(* IEC 61131-3 sources: LabBench/POU/04_AlarmAndSafety/FB, 5 files *)

(* ---- FB_DiagnosticScenario.st ---- *)
(*==============================================================================
    Название:    FB_DiagnosticScenario
    Автор:
    Дата:        2025-04-30
    Версия:      1.0

    Описание:    Функциональный блок обработки сценариев диагностики
                 Анализирует состояние системы на предмет обнаружения сценариев
                 неисправностей, таких как "насос работает, но нет расхода" и т.п.
==============================================================================*)
FUNCTION_BLOCK FB_DiagnosticScenario
VAR_INPUT
    (* Входные сигналы состояния системы *)

    (* Состояние насосов *)
    bPump1Running: BOOL;           (* Насос 1 работает *)
    bPump2Running: BOOL;           (* Насос 2 работает *)
    rPump1Speed: REAL;             (* Скорость насоса 1 (%) *)
    rPump2Speed: REAL;             (* Скорость насоса 2 (%) *)

    (* Состояние клапанов *)
    rPropValvePosition: REAL;      (* Положение пропорционального клапана (%) *)
    bEMValveOpen: BOOL;            (* Состояние электромагнитного клапана *)

    (* Состояние нагревателя *)
    bHeaterOn: BOOL;               (* Нагреватель включен *)
    rHeaterPower: REAL;            (* Мощность нагревателя (%) *)

    (* Сигналы с датчиков *)

    (* Давление *)
    rPressureKIE2: REAL;           (* Давление в емкости КИЕ2 (кПа) *)
    bPressureKIE2Valid: BOOL;      (* Сигнал валиден *)

    rPressurePipe: REAL;           (* Давление в трубопроводе (кПа) *)
    bPressurePipeValid: BOOL;      (* Сигнал валиден *)

    rPressurePumpIn1: REAL;        (* Давление перед насосом 1 (кПа) *)
    bPressurePumpIn1Valid: BOOL;   (* Сигнал валиден *)

    rPressurePumpOut1: REAL;       (* Давление после насоса 1 (кПа) *)
    bPressurePumpOut1Valid: BOOL;  (* Сигнал валиден *)

    rPressurePumpIn2: REAL;        (* Давление перед насосом 2 (кПа) *)
    bPressurePumpIn2Valid: BOOL;   (* Сигнал валиден *)

    rPressurePumpOut2: REAL;       (* Давление после насоса 2 (кПа) *)
    bPressurePumpOut2Valid: BOOL;  (* Сигнал валиден *)

    (* Расход *)
    rFlowPumpOut1: REAL;           (* Расход после насоса 1 (л/мин) *)
    bFlowPumpOut1Valid: BOOL;      (* Сигнал валиден *)

    rFlowPumpOut2: REAL;           (* Расход после насоса 2 (л/мин) *)
    bFlowPumpOut2Valid: BOOL;      (* Сигнал валиден *)

    rFlowPipe: REAL;               (* Расход в трубопроводе (л/мин) *)
    bFlowPipeValid: BOOL;          (* Сигнал валиден *)

    (* Уровень *)
    rLevelKIE1: REAL;              (* Уровень в емкости КИЕ1 (мм) *)
    bLevelKIE1Valid: BOOL;         (* Сигнал валиден *)

    bLevelLow: BOOL;               (* Уровень низкий (поплавок) *)
    bLevelMid: BOOL;               (* Уровень средний (поплавок) *)
    bLevelHigh: BOOL;              (* Уровень высокий (поплавок) *)
    bLevelValid: BOOL;             (* Сигналы валидны *)

    (* Температура *)
    rTemperature: REAL;            (* Температура (°C) *)
    bTemperatureValid: BOOL;       (* Сигнал валиден *)

    (* Управление *)
    bReset: BOOL;                  (* Сброс сценариев *)
    bEnable: BOOL := TRUE;         (* Разрешение работы *)
END_VAR

VAR_OUTPUT
    bAnyScenarioActive: BOOL;      (* Флаг наличия активных сценариев *)
    bBlockingRequired: BOOL;       (* Требуется блокировка *)
    bShutdownRequired: BOOL;       (* Требуется останов *)
    uiActiveScenarioCount: UINT;   (* Количество активных сценариев *)
    uiLastActiveScenarioIndex: UINT; (* Индекс последнего активного сценария *)
    dwActiveScenariosMask: DWORD;  (* Битовая маска активных сценариев *)
END_VAR

VAR
    (* Триггеры для обнаружения изменений *)
    rtPump1Running: R_TRIG;        (* Насос 1 запустился *)
    rtPump2Running: R_TRIG;        (* Насос 2 запустился *)
    rtHeaterOn: R_TRIG;            (* Нагреватель включился *)

    ftPump1Running: F_TRIG;        (* Насос 1 остановился *)
    ftPump2Running: F_TRIG;        (* Насос 2 остановился *)
    ftHeaterOn: F_TRIG;            (* Нагреватель выключился *)

    (* Таймеры для задержек обнаружения *)
    tonScenario1: TON;             (* Таймер для сценария 1 *)
    tonScenario2: TON;             (* Таймер для сценария 2 *)
    tonScenario3: TON;             (* Таймер для сценария 3 *)

    (* Локальные переменные *)
    uiCounter: UINT;               (* Счетчик для циклов *)

    (* Параметры сценариев *)
    rPump1DeltaP: REAL;            (* Перепад давления на насосе 1 *)
    rPump2DeltaP: REAL;            (* Перепад давления на насосе 2 *)

    (* Флаги обнаружения условий сценариев *)
    bPump1NoFlow: BOOL;            (* Условие "Насос 1 работает, но нет расхода" *)
    bPump2NoFlow: BOOL;            (* Условие "Насос 2 работает, но нет расхода" *)
    bPump1NoPressure: BOOL;        (* Условие "Насос 1 работает, но нет давления" *)
    bPump2NoPressure: BOOL;        (* Условие "Насос 2 работает, но нет давления" *)
    bPipeBlock: BOOL;              (* Условие "Блокировка в трубопроводе" *)
    bHeaterNoTempRise: BOOL;       (* Условие "Нагреватель включен, но температура не растет" *)
END_VAR

VAR CONSTANT
    (* Пороговые значения для обнаружения сценариев *)
    PUMP_MIN_SPEED: REAL := 10.0;          (* Минимальная скорость насоса (%) *)
    FLOW_THRESHOLD_LOW: REAL := 0.5;       (* Пороговое значение расхода (л/мин) *)
    PRESSURE_DELTA_MIN: REAL := 10.0;      (* Минимальный перепад давления (кПа) *)
    TEMPERATURE_RISE_MIN: REAL := 0.1;     (* Минимальный рост температуры (°C/мин) *)

    (* Времена задержек для обнаружения сценариев *)
    T_PUMP_NO_FLOW: TIME := T#5S;          (* Задержка для сценария "нет расхода" *)
    T_PUMP_NO_PRESSURE: TIME := T#3S;      (* Задержка для сценария "нет давления" *)
    T_HEATER_NO_TEMP: TIME := T#60S;       (* Задержка для сценария "нет роста температуры" *)
END_VAR

(* ======================================================================== *)
(* Основная логика функционального блока                                    *)
(* ======================================================================== *)

(* Обнаружение изменений состояния оборудования *)
rtPump1Running(CLK := bPump1Running);
rtPump2Running(CLK := bPump2Running);
rtHeaterOn(CLK := bHeaterOn);

ftPump1Running(CLK := bPump1Running);
ftPump2Running(CLK := bPump2Running);
ftHeaterOn(CLK := bHeaterOn);

(* Обработка команды сброса *)
IF bReset THEN
    (* Сброс всех сценариев *)
    FOR uiCounter := 1 TO MAX_SCENARIOS DO
        gaDiagScenarios[uiCounter].bActive := FALSE;
    END_FOR;

    (* Сброс таймеров *)
    tonScenario1(IN := FALSE);
    tonScenario2(IN := FALSE);
    tonScenario3(IN := FALSE);
END_IF;

(* Инициализация выходных переменных *)
bAnyScenarioActive := FALSE;
bBlockingRequired := FALSE;
bShutdownRequired := FALSE;
uiActiveScenarioCount := 0;
uiLastActiveScenarioIndex := 0;
dwActiveScenariosMask := 0;

(* ======================================================================== *)
(* Обнаружение условий для сценариев                                        *)
(* ======================================================================== *)

IF bEnable THEN

    (* Расчет параметров системы *)
    IF bPressurePumpIn1Valid AND bPressurePumpOut1Valid THEN
        rPump1DeltaP := rPressurePumpOut1 - rPressurePumpIn1;
    ELSE
        rPump1DeltaP := 0.0;
    END_IF;

    IF bPressurePumpIn2Valid AND bPressurePumpOut2Valid THEN
        rPump2DeltaP := rPressurePumpOut2 - rPressurePumpIn2;
    ELSE
        rPump2DeltaP := 0.0;
    END_IF;

    (* Условие "Насос 1 работает, но нет расхода" *)
    bPump1NoFlow := bPump1Running AND rPump1Speed > PUMP_MIN_SPEED AND
                    bFlowPumpOut1Valid AND rFlowPumpOut1 < FLOW_THRESHOLD_LOW;

    (* Условие "Насос 2 работает, но нет расхода" *)
    bPump2NoFlow := bPump2Running AND rPump2Speed > PUMP_MIN_SPEED AND
                    bFlowPumpOut2Valid AND rFlowPumpOut2 < FLOW_THRESHOLD_LOW;

    (* Условие "Насос 1 работает, но нет давления" *)
    bPump1NoPressure := bPump1Running AND rPump1Speed > PUMP_MIN_SPEED AND
                        bPressurePumpIn1Valid AND bPressurePumpOut1Valid AND
                        rPump1DeltaP < PRESSURE_DELTA_MIN;

    (* Условие "Насос 2 работает, но нет давления" *)
    bPump2NoPressure := bPump2Running AND rPump2Speed > PUMP_MIN_SPEED AND
                        bPressurePumpIn2Valid AND bPressurePumpOut2Valid AND
                        rPump2DeltaP < PRESSURE_DELTA_MIN;

    (* Условие "Блокировка в трубопроводе" *)
    bPipeBlock := bFlowPipeValid AND rFlowPipe < FLOW_THRESHOLD_LOW AND
                  bPressurePipeValid AND rPressurePipe > (rPressureKIE2 * 1.5);

    (* Условие "Нагреватель включен, но температура не растет" *)
    (* Требует дополнительной логики с отслеживанием изменения температуры во времени *)
    bHeaterNoTempRise := FALSE; (* Пока не реализовано *)

    (* ======================================================================== *)
    (* Обработка таймеров задержки обнаружения сценариев                       *)
    (* ======================================================================== *)

    (* Таймер для сценария "Насос 1 работает, но нет расхода" *)
    tonScenario1(IN := bPump1NoFlow, PT := T_PUMP_NO_FLOW);

    (* Таймер для сценария "Насос 2 работает, но нет расхода" *)
    tonScenario2(IN := bPump2NoFlow, PT := T_PUMP_NO_FLOW);

    (* Таймер для сценария "Нагреватель включен, но температура не растет" *)
    tonScenario3(IN := bHeaterNoTempRise, PT := T_HEATER_NO_TEMP);

    (* ======================================================================== *)
    (* Активация сценариев диагностики                                         *)
    (* ======================================================================== *)

    (* Сценарий 1: "Насос 1 работает, но нет расхода" *)
    IF tonScenario1.Q THEN
        gaDiagScenarios[1].bActive := TRUE;
        gaDiagScenarios[1].eType := DIAG_PUMP_NO_FLOW;
        gaDiagScenarios[1].wSourceID := PUMP1_ID;
        gaDiagScenarios[1].wDeviceID := PUMP1_ID;
        gaDiagScenarios[1].eBlockingLevel := DEVICE_BLOCKING;
        gaDiagScenarios[1].bRequireShutdown := FALSE;
        gaDiagScenarios[1].rValue1 := rPump1Speed;
        gaDiagScenarios[1].rValue2 := rFlowPumpOut1;
        gaDiagScenarios[1].wErrorCode := 16#0101;
        gaDiagScenarios[1].sMessage := 'Насос 1 работает, но нет расхода';
    END_IF;

    (* Сценарий 2: "Насос 2 работает, но нет расхода" *)
    IF tonScenario2.Q THEN
        gaDiagScenarios[2].bActive := TRUE;
        gaDiagScenarios[2].eType := DIAG_PUMP_NO_FLOW;
        gaDiagScenarios[2].wSourceID := PUMP2_ID;
        gaDiagScenarios[2].wDeviceID := PUMP2_ID;
        gaDiagScenarios[2].eBlockingLevel := DEVICE_BLOCKING;
        gaDiagScenarios[2].bRequireShutdown := FALSE;
        gaDiagScenarios[2].rValue1 := rPump2Speed;
        gaDiagScenarios[2].rValue2 := rFlowPumpOut2;
        gaDiagScenarios[2].wErrorCode := 16#0102;
        gaDiagScenarios[2].sMessage := 'Насос 2 работает, но нет расхода';
    END_IF;

    (* Сценарий 3: "Насос 1 работает, но нет давления" *)
    IF bPump1NoPressure THEN
        gaDiagScenarios[3].bActive := TRUE;
        gaDiagScenarios[3].eType := DIAG_PUMP_NO_PRESSURE;
        gaDiagScenarios[3].wSourceID := PUMP1_ID;
        gaDiagScenarios[3].wDeviceID := PUMP1_ID;
        gaDiagScenarios[3].eBlockingLevel := DEVICE_BLOCKING;
        gaDiagScenarios[3].bRequireShutdown := FALSE;
        gaDiagScenarios[3].rValue1 := rPump1Speed;
        gaDiagScenarios[3].rValue2 := rPump1DeltaP;
        gaDiagScenarios[3].wErrorCode := 16#0103;
        gaDiagScenarios[3].sMessage := 'Насос 1 работает, но нет давления';
    END_IF;

    (* Сценарий 4: "Насос 2 работает, но нет давления" *)
    IF bPump2NoPressure THEN
        gaDiagScenarios[4].bActive := TRUE;
        gaDiagScenarios[4].eType := DIAG_PUMP_NO_PRESSURE;
        gaDiagScenarios[4].wSourceID := PUMP2_ID;
        gaDiagScenarios[4].wDeviceID := PUMP2_ID;
        gaDiagScenarios[4].eBlockingLevel := DEVICE_BLOCKING;
        gaDiagScenarios[4].bRequireShutdown := FALSE;
        gaDiagScenarios[4].rValue1 := rPump2Speed;
        gaDiagScenarios[4].rValue2 := rPump2DeltaP;
        gaDiagScenarios[4].wErrorCode := 16#0104;
        gaDiagScenarios[4].sMessage := 'Насос 2 работает, но нет давления';
    END_IF;

    (* Сценарий 5: "Блокировка в трубопроводе" *)
    IF bPipeBlock THEN
        gaDiagScenarios[5].bActive := TRUE;
        gaDiagScenarios[5].eType := DIAG_PIPE_BLOCK;
        gaDiagScenarios[5].wSourceID := SYSTEM_ID;
        gaDiagScenarios[5].wDeviceID := 0;
        gaDiagScenarios[5].eBlockingLevel := SYSTEM_BLOCKING;
        gaDiagScenarios[5].bRequireShutdown := TRUE;
        gaDiagScenarios[5].rValue1 := rFlowPipe;
        gaDiagScenarios[5].rValue2 := rPressurePipe;
        gaDiagScenarios[5].wErrorCode := 16#0105;
        gaDiagScenarios[5].sMessage := 'Блокировка в трубопроводе';
    END_IF;

    (* Сценарий 6: "Нагреватель включен, но температура не растет" *)
    IF tonScenario3.Q THEN
        gaDiagScenarios[6].bActive := TRUE;
        gaDiagScenarios[6].eType := DIAG_HEATER_NO_TEMP_RISE;
        gaDiagScenarios[6].wSourceID := HEATER_ID;
        gaDiagScenarios[6].wDeviceID := HEATER_ID;
        gaDiagScenarios[6].eBlockingLevel := DEVICE_BLOCKING;
        gaDiagScenarios[6].bRequireShutdown := FALSE;
        gaDiagScenarios[6].rValue1 := rHeaterPower;
        gaDiagScenarios[6].rValue2 := rTemperature;
        gaDiagScenarios[6].wErrorCode := 16#0106;
        gaDiagScenarios[6].sMessage := 'Нагреватель включен, но температура не растет';
    END_IF;

    (* ======================================================================== *)
    (* Обработка результатов анализа сценариев                                 *)
    (* ======================================================================== *)

    (* Обработка всех сценариев *)
    FOR uiCounter := 1 TO MAX_SCENARIOS DO
        IF gaDiagScenarios[uiCounter].bActive THEN
            (* Сценарий активен *)
            bAnyScenarioActive := TRUE;
            uiActiveScenarioCount := uiActiveScenarioCount + 1;
            uiLastActiveScenarioIndex := uiCounter;

            (* Установка бита в маске активных сценариев (только для первых 32 сценариев) *)
            IF uiCounter <= 32 THEN
                dwActiveScenariosMask := dwActiveScenariosMask OR SHL(DWORD#1, uiCounter-1);
            END_IF;

            (* Проверка требований блокировки и останова *)
            IF gaDiagScenarios[uiCounter].eBlockingLevel <> NO_BLOCKING THEN
                bBlockingRequired := TRUE;
            END_IF;

            IF gaDiagScenarios[uiCounter].bRequireShutdown THEN
                bShutdownRequired := TRUE;
            END_IF;
        END_IF;
    END_FOR;
END_IF;

(* ---- FB_ErrorManager.st ---- *)
(*==============================================================================
    Название:    FB_ErrorManager
    Автор:
    Дата:        2025-04-28
    Версия:      1.0

    Описание:    Функциональный блок управления ошибками и блокировками
                 Обрабатывает ошибки различных категорий, управляет блокировками
                 оборудования и формирует сигналы для сигнальной лампы
==============================================================================*)
FUNCTION_BLOCK FB_ErrorManager
VAR_INPUT
    bResetAll: BOOL;                      (* Общий сброс всех ошибок *)
    bResetMeasurement: BOOL;              (* Сброс ошибок измерительной системы *)
    bResetPropValve: BOOL;                (* Сброс ошибок пропорционального клапана *)
    bResetEMValve: BOOL;                  (* Сброс ошибок электромагнитного клапана *)
    bResetPump1: BOOL;                    (* Сброс ошибок насоса 1 *)
    bResetPump2: BOOL;                    (* Сброс ошибок насоса 2 *)
END_VAR

VAR_OUTPUT
    bAnyError: BOOL;                      (* Флаг наличия любых ошибок *)
    bSystemBlocking: BOOL;                (* Флаг полной блокировки системы *)
    eLampMode: E_LampBlinkMode;           (* Режим работы сигнальной лампы *)
    dwActiveErrorMask: DWORD;             (* Битовая маска активных ошибок *)

    (* Блокировки устройств *)
    bPropValveBlocking: BOOL;             (* Блокировка пропорционального клапана *)
    bEMValveBlocking: BOOL;               (* Блокировка электромагнитного клапана *)
    bPump1Blocking: BOOL;                 (* Блокировка насоса 1 *)
    bPump2Blocking: BOOL;                 (* Блокировка насоса 2 *)
END_VAR

VAR
    (* Локальные переменные *)
    uiCounter: UINT;                      (* Счетчик для циклов *)
    bHasErrorCategory: ARRAY[0..4] OF BOOL; (* Флаги наличия ошибок по категориям *)
END_VAR

(* ======================================================================== *)
(* Основная логика функционального блока                                    *)
(* ======================================================================== *)

(* Обработка команд сброса ошибок *)
IF bResetAll THEN
    (* Сброс всех ошибок *)
    FOR uiCounter := 1 TO MAX_ERRORS DO
        gaBlockingErrors[uiCounter].bActive := FALSE;
    END_FOR;
ELSE
    (* Выборочный сброс ошибок *)
    IF bResetMeasurement THEN
        (* Сброс ошибок измерительной системы *)
        FOR uiCounter := 1 TO MAX_ERRORS DO
            IF gaBlockingErrors[uiCounter].eCategory = ERROR_MEASUREMENT THEN
                gaBlockingErrors[uiCounter].bActive := FALSE;
            END_IF;
        END_FOR;
    END_IF;

    IF bResetPropValve THEN
        (* Сброс ошибок пропорционального клапана *)
        FOR uiCounter := 1 TO MAX_ERRORS DO
            IF gaBlockingErrors[uiCounter].wDeviceID = PROP_VALVE_ID THEN
                gaBlockingErrors[uiCounter].bActive := FALSE;
            END_IF;
        END_FOR;
    END_IF;

    IF bResetEMValve THEN
        (* Сброс ошибок электромагнитного клапана *)
        FOR uiCounter := 1 TO MAX_ERRORS DO
            IF gaBlockingErrors[uiCounter].wDeviceID = EM_VALVE_ID THEN
                gaBlockingErrors[uiCounter].bActive := FALSE;
            END_IF;
        END_FOR;
    END_IF;

    IF bResetPump1 THEN
        (* Сброс ошибок насоса 1 *)
        FOR uiCounter := 1 TO MAX_ERRORS DO
            IF gaBlockingErrors[uiCounter].wDeviceID = PUMP1_ID THEN
                gaBlockingErrors[uiCounter].bActive := FALSE;
            END_IF;
        END_FOR;
    END_IF;

    IF bResetPump2 THEN
        (* Сброс ошибок насоса 2 *)
        FOR uiCounter := 1 TO MAX_ERRORS DO
            IF gaBlockingErrors[uiCounter].wDeviceID = PUMP2_ID THEN
                gaBlockingErrors[uiCounter].bActive := FALSE;
            END_IF;
        END_FOR;
    END_IF;
END_IF;

(* Сброс флагов *)
bAnyError := FALSE;
bSystemBlocking := FALSE;
dwActiveErrorMask := 0;
bPropValveBlocking := FALSE;
bEMValveBlocking := FALSE;
bPump1Blocking := FALSE;
bPump2Blocking := FALSE;

(* Сброс флагов категорий ошибок *)
FOR uiCounter := 0 TO 4 DO
    bHasErrorCategory[uiCounter] := FALSE;
END_FOR;

(* Обработка всех ошибок *)
FOR uiCounter := 1 TO MAX_ERRORS DO
    IF gaBlockingErrors[uiCounter].bActive THEN
        (* Ошибка активна *)
        bAnyError := TRUE;

        (* Установка бита в маске активных ошибок (только для первых 32 ошибок) *)
        IF uiCounter <= 32 THEN
            dwActiveErrorMask := dwActiveErrorMask OR SHL(DWORD#1, uiCounter-1);
        END_IF;

        (* Отметка категории ошибки *)
        bHasErrorCategory[ENUM_TO_DINT(gaBlockingErrors[uiCounter].eCategory)] := TRUE;

        (* Обработка блокировок *)
        CASE gaBlockingErrors[uiCounter].eBlockingLevel OF
            SYSTEM_BLOCKING:
                (* Полная блокировка системы *)
                bSystemBlocking := TRUE;

            DEVICE_BLOCKING:
                (* Блокировка конкретного устройства *)
                CASE gaBlockingErrors[uiCounter].wDeviceID OF
                    PROP_VALVE_ID:
                        bPropValveBlocking := TRUE;

                    EM_VALVE_ID:
                        bEMValveBlocking := TRUE;

                    PUMP1_ID:
                        bPump1Blocking := TRUE;

                    PUMP2_ID:
                        bPump2Blocking := TRUE;
                END_CASE;
        END_CASE;
    END_IF;
END_FOR;

(* Определение режима работы сигнальной лампы *)
IF bAnyError THEN
    IF bHasErrorCategory[ENUM_TO_DINT(ERROR_MEASUREMENT)] THEN
        (* Ошибка измерения - быстрое мигание *)
        eLampMode := LAMP_FAST;
    ELSIF bHasErrorCategory[ENUM_TO_DINT(ERROR_COMMUNICATION)] THEN
        (* Ошибка связи - медленное мигание *)
        eLampMode := LAMP_SLOW;
    ELSIF bHasErrorCategory[ENUM_TO_DINT(ERROR_EQUIPMENT)] THEN
        (* Ошибка оборудования - постоянно горит *)
        eLampMode := LAMP_ON;
    ELSIF bHasErrorCategory[ENUM_TO_DINT(ERROR_PROCESS)] THEN
        (* Ошибка процесса - быстрое мигание *)
        eLampMode := LAMP_FAST;
    ELSE
        (* Неизвестная ошибка - постоянно горит *)
        eLampMode := LAMP_ON;
    END_IF;
ELSE
    (* Нет ошибок - лампа выключена *)
    eLampMode := LAMP_OFF;
END_IF;

(* ---- FB_LampController.st ---- *)
(*==============================================================================
    Название:    FB_LampController
    Автор:
    Дата:        2025-04-28
    Версия:      1.1

    Описание:    Функциональный блок управления сигнальной лампой
                 Генерирует сигналы для различных режимов работы лампы

                 Реализован как level-controlled (LCon) блок
==============================================================================*)
FUNCTION_BLOCK FB_LampController (* LCon *)
VAR_INPUT
    eMode: E_LampBlinkMode;               (* Режим работы лампы *)
    bEnable: BOOL := TRUE;                (* Разрешение работы *)
END_VAR

VAR_OUTPUT
    bOutput: BOOL;                        (* Выходной сигнал *)
END_VAR

VAR
    (* Таймеры для различных режимов мигания *)
    tonSlow: TON;                         (* Таймер медленного мигания (1 Гц) *)
    tonFast: TON;                         (* Таймер быстрого мигания (4 Гц) *)

    (* Состояния для различных режимов *)
    bSlowState: BOOL;                     (* Состояние медленного мигания *)
    bFastState: BOOL;                     (* Состояние быстрого мигания *)
END_VAR

VAR CONSTANT
    (* Константы времени для различных режимов *)
    T_SLOW: TIME := T#500MS;              (* Период для медленного мигания - 1 Гц *)
    T_FAST: TIME := T#125MS;              (* Период для быстрого мигания - 4 Гц *)
END_VAR

(* ======================================================================== *)
(* Основная логика функционального блока                                    *)
(* ======================================================================== *)

(* Генерация сигналов для различных режимов мигания *)
(* Медленное мигание - 1 Гц *)
tonSlow(IN := NOT tonSlow.Q, PT := T_SLOW);
IF tonSlow.Q THEN
    bSlowState := NOT bSlowState;
END_IF;

(* Быстрое мигание - 4 Гц *)
tonFast(IN := NOT tonFast.Q, PT := T_FAST);
IF tonFast.Q THEN
    bFastState := NOT bFastState;
END_IF;

(* Выбор режима мигания *)
IF bEnable THEN
    CASE eMode OF
        LAMP_OFF:
            bOutput := FALSE;

        LAMP_ON:
            bOutput := TRUE;

        LAMP_SLOW:
            bOutput := bSlowState;

        LAMP_FAST:
            bOutput := bFastState;

        ELSE
            (* По умолчанию - выключено *)
            bOutput := FALSE;
    END_CASE;
ELSE
    (* При отключенном блоке - выходной сигнал выключен *)
    bOutput := FALSE;
END_IF;

(* ---- FB_ShutdownSequencer.st ---- *)
(*==============================================================================
    Название:    FB_ShutdownSequencer
    Автор:
    Дата:        2025-04-30
    Версия:      1.0

    Описание:    Функциональный блок для управления последовательностью останова
                 Обеспечивает правильный порядок выключения оборудования
                 в штатном и аварийном режимах
==============================================================================*)
FUNCTION_BLOCK FB_ShutdownSequencer
VAR_IN_OUT
    stSequence: ST_ShutdownSequence;   (* Структура данных последовательности останова *)
END_VAR

VAR_INPUT
    bStartNormal: BOOL;                (* Запуск нормального останова *)
    bStartEmergency: BOOL;             (* Запуск аварийного останова *)
    bReset: BOOL;                      (* Сброс последовательности *)

    (* Состояние оборудования *)
    bHeaterOn: BOOL;                   (* Нагреватель включен *)
    rPump1Speed: REAL;                 (* Скорость насоса 1 (%) *)
    rPump2Speed: REAL;                 (* Скорость насоса 2 (%) *)
    rPropValvePosition: REAL;          (* Положение пропорционального клапана (%) *)
    bEMValveOpen: BOOL;                (* Состояние электромагнитного клапана *)
END_VAR

VAR_OUTPUT
    (* Команды управления оборудованием *)
    bHeaterOff: BOOL;                  (* Команда выключения нагревателя *)
    rPump1SpeedSetpoint: REAL;         (* Задание скорости насоса 1 (%) *)
    rPump2SpeedSetpoint: REAL;         (* Задание скорости насоса 2 (%) *)
    bPump1Stop: BOOL;                  (* Команда остановки насоса 1 *)
    bPump2Stop: BOOL;                  (* Команда остановки насоса 2 *)
    rPropValveSetpoint: REAL;          (* Задание положения пропорционального клапана (%) *)
    bEMValveClose: BOOL;               (* Команда закрытия электромагнитного клапана *)
END_VAR

VAR
    (* Триггеры *)
    rtStartNormal: R_TRIG;             (* Триггер запуска нормального останова *)
    rtStartEmergency: R_TRIG;          (* Триггер запуска аварийного останова *)
    rtReset: R_TRIG;                   (* Триггер сброса *)

    (* Таймеры *)
    tonStep: TON;                      (* Таймер текущего шага *)
    tonTimeout: TON;                   (* Таймер таймаута *)

    (* Локальные переменные *)
    tCurrentTime: TIME;                (* Текущее время *)
    tElapsedTime: TIME;                (* Прошедшее время *)
    rRateCalc: REAL;                   (* Расчетная скорость изменения *)
END_VAR

(* ======================================================================== *)
(* Основная логика функционального блока                                    *)
(* ======================================================================== *)

(* Обработка триггеров *)
rtStartNormal(CLK := bStartNormal);
rtStartEmergency(CLK := bStartEmergency);
rtReset(CLK := bReset);

(* Запуск последовательности останова *)
IF rtStartNormal.Q OR rtStartEmergency.Q THEN
    (* Инициализация последовательности *)
    stSequence.eCurrentStep := SHUTDOWN_INIT;
    stSequence.bInProgress := TRUE;
    stSequence.bEmergency := rtStartEmergency.Q;
    stSequence.bCompleted := FALSE;
    stSequence.bError := FALSE;
    stSequence.tStepStartTime := T#0S;

    (* Сброс таймеров *)
    tonStep(IN := FALSE);
    tonTimeout(IN := FALSE);
END_IF;

(* Сброс последовательности *)
IF rtReset.Q THEN
    (* Сброс всех параметров *)
    stSequence.eCurrentStep := SHUTDOWN_INIT;
    stSequence.bInProgress := FALSE;
    stSequence.bEmergency := FALSE;
    stSequence.bCompleted := FALSE;
    stSequence.bError := FALSE;
    stSequence.tStepStartTime := T#0S;

    (* Сброс таймеров *)
    tonStep(IN := FALSE);
    tonTimeout(IN := FALSE);

    (* Сброс выходов *)
    bHeaterOff := FALSE;
    rPump1SpeedSetpoint := 100.0;
    rPump2SpeedSetpoint := 100.0;
    bPump1Stop := FALSE;
    bPump2Stop := FALSE;
    rPropValveSetpoint := 100.0;
    bEMValveClose := FALSE;

    RETURN;
END_IF;

(* Обработка последовательности останова *)
IF stSequence.bInProgress THEN
    (* Отработка шагов последовательности *)
    CASE stSequence.eCurrentStep OF
        SHUTDOWN_INIT:
            (* Инициализация последовательности *)
            stSequence.tStepStartTime := T#0S;
            bHeaterOff := FALSE;
            bPump1Stop := FALSE;
            bPump2Stop := FALSE;
            bEMValveClose := FALSE;

            (* Переход к следующему шагу *)
            stSequence.eCurrentStep := SHUTDOWN_HEATER_OFF;

        SHUTDOWN_HEATER_OFF:
            (* Выключение нагревателя *)
            bHeaterOff := TRUE;

            (* Проверка выполнения шага *)
            IF NOT bHeaterOn THEN
                (* Нагреватель выключен - переход к следующему шагу *)
                stSequence.eCurrentStep := SHUTDOWN_PUMP_SLOWDOWN;
                tonStep(IN := FALSE);
            ELSE
                (* Ожидание выключения с таймаутом *)
                tonStep(IN := TRUE, PT := stSequence.tHeaterOffTimeout);
                IF tonStep.Q THEN
                    (* Таймаут - переход к следующему шагу с ошибкой *)
                    stSequence.eCurrentStep := SHUTDOWN_PUMP_SLOWDOWN;
                    stSequence.bError := TRUE;
                    tonStep(IN := FALSE);
                END_IF;
            END_IF;

        SHUTDOWN_PUMP_SLOWDOWN:
            (* Снижение скорости насосов *)
            IF stSequence.bEmergency THEN
                (* Аварийный останов - сразу к остановке насосов *)
                stSequence.eCurrentStep := SHUTDOWN_PUMP_STOP;
            ELSE
                (* Плавное снижение скорости насосов *)
                tonStep(IN := TRUE, PT := stSequence.tPumpSlowdownTime);

                (* Расчет скорости с учетом прошедшего времени *)
                rRateCalc := 100.0 - (TIME_TO_REAL(tonStep.ET) / TIME_TO_REAL(stSequence.tPumpSlowdownTime)) * 100.0;

                (* Установка скорости насосов *)
                rPump1SpeedSetpoint := MAX(0.0, rRateCalc);
                rPump2SpeedSetpoint := MAX(0.0, rRateCalc);

                (* Проверка завершения шага *)
                IF tonStep.Q THEN
                    (* Снижение скорости завершено - переход к остановке насосов *)
                    stSequence.eCurrentStep := SHUTDOWN_PUMP_STOP;
                    tonStep(IN := FALSE);
                END_IF;
            END_IF;

        SHUTDOWN_PUMP_STOP:
            (* Полная остановка насосов *)
            bPump1Stop := TRUE;
            bPump2Stop := TRUE;
            rPump1SpeedSetpoint := 0.0;
            rPump2SpeedSetpoint := 0.0;

            (* Проверка выполнения шага *)
            IF rPump1Speed <= 0.1 AND rPump2Speed <= 0.1 THEN
                (* Насосы остановлены - переход к следующему шагу *)
                stSequence.eCurrentStep := SHUTDOWN_VALVE_CLOSE;
                tonStep(IN := FALSE);
            ELSE
                (* Ожидание остановки с таймаутом *)
                tonStep(IN := TRUE, PT := stSequence.tPumpStopTimeout);
                IF tonStep.Q THEN
                    (* Таймаут - переход к следующему шагу с ошибкой *)
                    stSequence.eCurrentStep := SHUTDOWN_VALVE_CLOSE;
                    stSequence.bError := TRUE;
                    tonStep(IN := FALSE);
                END_IF;
            END_IF;

        SHUTDOWN_VALVE_CLOSE:
            (* Закрытие клапанов *)
            bEMValveClose := TRUE;

            IF stSequence.bEmergency THEN
                (* Аварийный останов - сразу закрываем пропорциональный клапан *)
                rPropValveSetpoint := 0.0;
            ELSE
                (* Плавное закрытие пропорционального клапана *)
                tonStep(IN := TRUE, PT := stSequence.tValveCloseTimeout);

                (* Расчет положения с учетом прошедшего времени *)
                rRateCalc := 100.0 - (TIME_TO_REAL(tonStep.ET) / TIME_TO_REAL(stSequence.tValveCloseTimeout)) * 100.0;

                (* Установка положения клапана *)
                rPropValveSetpoint := MAX(0.0, rRateCalc);
            END_IF;

            (* Проверка выполнения шага *)
            IF rPropValvePosition <= 0.1 AND NOT bEMValveOpen THEN
                (* Клапаны закрыты - переход к следующему шагу *)
                stSequence.eCurrentStep := SHUTDOWN_WAIT;
                tonStep(IN := FALSE);
            ELSE
                (* Ожидание закрытия с таймаутом *)
                tonStep(IN := TRUE, PT := stSequence.tValveCloseTimeout);
                IF tonStep.Q THEN
                    (* Таймаут - переход к следующему шагу с ошибкой *)
                    stSequence.eCurrentStep := SHUTDOWN_WAIT;
                    stSequence.bError := TRUE;
                    tonStep(IN := FALSE);
                END_IF;
            END_IF;

        SHUTDOWN_WAIT:
            (* Ожидание перед завершением останова *)
            tonStep(IN := TRUE, PT := stSequence.tWaitTime);

            (* Проверка выполнения шага *)
            IF tonStep.Q THEN
                (* Ожидание завершено - переход к завершению останова *)
                stSequence.eCurrentStep := SHUTDOWN_COMPLETE;
                tonStep(IN := FALSE);
            END_IF;

        SHUTDOWN_COMPLETE:
            (* Останов завершен *)
            stSequence.bInProgress := FALSE;
            stSequence.bCompleted := TRUE;

            (* Финальная проверка состояния оборудования *)
            IF bHeaterOn OR rPump1Speed > 0.1 OR rPump2Speed > 0.1 OR
               rPropValvePosition > 0.1 OR bEMValveOpen THEN
                (* Не все оборудование остановлено - ошибка *)
                stSequence.bError := TRUE;
                stSequence.eCurrentStep := SHUTDOWN_ERROR;
            END_IF;

        SHUTDOWN_ERROR:
            (* Ошибка останова - ничего не делаем, ждем сброса *)
            stSequence.bInProgress := FALSE;
            stSequence.bError := TRUE;
    END_CASE;
ELSE
    (* Последовательность неактивна - сброс выходов *)
    IF NOT stSequence.bCompleted THEN
        bHeaterOff := FALSE;
        rPump1SpeedSetpoint := 100.0;
        rPump2SpeedSetpoint := 100.0;
        bPump1Stop := FALSE;
        bPump2Stop := FALSE;
        rPropValveSetpoint := 100.0;
        bEMValveClose := FALSE;
    END_IF;
END_IF;

(* ---- FB_SystemManager.st ---- *)
(*==============================================================================
    Название:    FB_SystemManager
    Автор:
    Дата:        2025-04-30
    Версия:      1.0

    Описание:    Функциональный блок управления состоянием системы
                 Координирует работу всей диагностической системы,
                 обрабатывает ошибки и сценарии, управляет блокировками
                 и последовательностью останова
==============================================================================*)
FUNCTION_BLOCK FB_SystemManager
VAR_INPUT
    (* Состояние системы *)
    bSystemInitialized: BOOL;         (* Система инициализирована *)
    bAnyError: BOOL;                  (* Флаг наличия ошибок *)
    bAnyScenarioActive: BOOL;         (* Флаг наличия активных сценариев *)
    bAnyBlockingRequired: BOOL;       (* Требуется блокировка *)
    bAnyShutdownRequired: BOOL;       (* Требуется останов *)

    (* Состояние последовательности останова *)
    bShutdownInProgress: BOOL;        (* Последовательность останова активна *)
    bShutdownCompleted: BOOL;         (* Останов завершен *)
    bShutdownError: BOOL;             (* Ошибка в процессе останова *)

    (* Команды управления *)
    bResetSystem: BOOL;               (* Сброс системы *)
    bStartNormalShutdown: BOOL;       (* Запуск нормального останова *)
    bStartEmergencyShutdown: BOOL;    (* Запуск аварийного останова *)
END_VAR

VAR_OUTPUT
    eSystemState: E_SystemState;      (* Текущее состояние системы *)
    bSystemBlockingRequired: BOOL;    (* Требуется блокировка системы *)
    bSystemShutdownRequired: BOOL;    (* Требуется останов системы *)
    bSystemResetRequired: BOOL;       (* Требуется сброс системы *)
END_VAR

VAR
    (* Триггеры *)
    rtResetSystem: R_TRIG;            (* Триггер сброса системы *)
    rtStartNormalShutdown: R_TRIG;    (* Триггер запуска нормального останова *)
    rtStartEmergencyShutdown: R_TRIG; (* Триггер запуска аварийного останова *)

    (* Текущее состояние *)
    ePrevSystemState: E_SystemState;  (* Предыдущее состояние системы *)
    tStateChangeTime: TON;            (* Таймер для измерения времени в состоянии *)
END_VAR

(* ======================================================================== *)
(* Основная логика функционального блока                                    *)
(* ======================================================================== *)

(* Обработка триггеров *)
rtResetSystem(CLK := bResetSystem);
rtStartNormalShutdown(CLK := bStartNormalShutdown);
rtStartEmergencyShutdown(CLK := bStartEmergencyShutdown);

(* Сохранение предыдущего состояния *)
IF eSystemState <> ePrevSystemState THEN
    ePrevSystemState := eSystemState;
    tStateChangeTime(IN := FALSE);
END_IF;

(* Запуск таймера состояния *)
tStateChangeTime(IN := TRUE, PT := T#24H); (* 24 часа - фактически бесконечность для таймера *)

(* Определение текущего состояния системы *)
IF NOT bSystemInitialized THEN
    (* Система не инициализирована *)
    eSystemState := SYSTEM_INIT;
    bSystemBlockingRequired := FALSE;
    bSystemShutdownRequired := FALSE;
    bSystemResetRequired := FALSE;

ELSIF bShutdownInProgress THEN
    (* Выполняется последовательность останова *)
    IF bAnyError OR bAnyBlockingRequired OR bAnyShutdownRequired THEN
        (* Аварийный останов *)
        eSystemState := SYSTEM_ERROR_SHUTDOWN;
    ELSE
        (* Нормальный останов *)
        eSystemState := SYSTEM_SHUTDOWN;
    END_IF;

    bSystemBlockingRequired := TRUE;
    bSystemShutdownRequired := TRUE;
    bSystemResetRequired := FALSE;

ELSIF bShutdownCompleted THEN
    (* Останов завершен *)
    IF bShutdownError OR bAnyError OR bAnyBlockingRequired THEN
        (* Останов с ошибкой *)
        eSystemState := SYSTEM_ERROR;
        bSystemBlockingRequired := TRUE;
        bSystemShutdownRequired := FALSE;
        bSystemResetRequired := TRUE;
    ELSE
        (* Нормальный останов *)
        eSystemState := SYSTEM_READY;
        bSystemBlockingRequired := FALSE;
        bSystemShutdownRequired := FALSE;
        bSystemResetRequired := FALSE;
    END_IF;

ELSIF bAnyError OR bAnyBlockingRequired THEN
    (* Ошибка в системе *)
    eSystemState := SYSTEM_ERROR;
    bSystemBlockingRequired := TRUE;

    (* Требуется ли останов *)
    bSystemShutdownRequired := bAnyShutdownRequired;
    bSystemResetRequired := TRUE;

ELSIF bAnyScenarioActive THEN
    (* Активен сценарий, но без блокировки *)
    eSystemState := SYSTEM_RUNNING;
    bSystemBlockingRequired := FALSE;
    bSystemShutdownRequired := bAnyShutdownRequired;
    bSystemResetRequired := FALSE;

ELSE
    (* Нормальная работа *)
    eSystemState := SYSTEM_RUNNING;
    bSystemBlockingRequired := FALSE;
    bSystemShutdownRequired := FALSE;
    bSystemResetRequired := FALSE;
END_IF;

(* Обработка команд *)
IF rtResetSystem.Q THEN
    (* Сброс системы *)
    IF eSystemState = SYSTEM_ERROR AND NOT bShutdownInProgress THEN
        (* Можно выполнить сброс только в состоянии ошибки и не во время останова *)
        eSystemState := SYSTEM_READY;
        bSystemBlockingRequired := FALSE;
        bSystemShutdownRequired := FALSE;
        bSystemResetRequired := FALSE;
    END_IF;
END_IF;

(* Команды запуска останова имеют приоритет *)
IF rtStartEmergencyShutdown.Q OR rtStartNormalShutdown.Q THEN
    (* Запуск останова *)
    IF rtStartEmergencyShutdown.Q THEN
        eSystemState := SYSTEM_ERROR_SHUTDOWN;
    ELSE
        eSystemState := SYSTEM_SHUTDOWN;
    END_IF;

    bSystemBlockingRequired := TRUE;
    bSystemShutdownRequired := TRUE;
    bSystemResetRequired := FALSE;
END_IF;
